FUNCTION_BLOCK FB_SomeGrantryRobot
VAR_INPUT
END_VAR
VAR_OUTPUT
END_VAR
VAR
END_VAR

END_FUNCTION_BLOCK

(* stored: Version 1.1.0.1, ProductVersion 3.1.4024.9
   POU FB_SomeGrantryRobot: Id {8623795a-912a-40c2-a294-dc497aee4ac5}, SpecialFunc None *)
